% RSLogix 500 project Flip-Flop.RSS, saved by version 8.30.01.01 %
PROJECT "UNTITLED"    % processor: Bul.1763 MicroLogix 1100 Series A %

PROGRAM FILES
  LAD 2   4 rungs

DATA FILES
  O0 OUTPUT  4 elements
  I1 INPUT  6 elements
  S2 STATUS  66 elements
  B3 BINARY  1 elements
  T4 TIMER  2 elements
  C5 COUNTER  1 elements
  R6 CONTROL  1 elements
  N7 INTEGER  1 elements
  F8 FLOAT  1 elements

LADDER 2
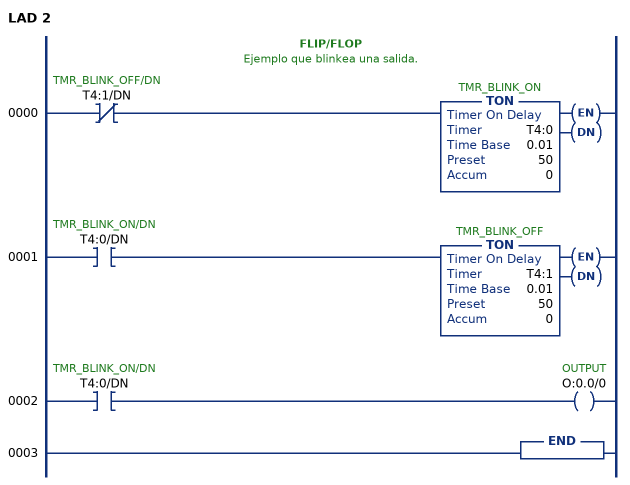
% Rung: 0 %  % edit flag set %
% TITLE: FLIP/FLOP %
% Ejemplo que blinkea una salida. %
SOR XIO T4:1/DN TON T4:0 0.01 50 0 EOR
%   T4:1  TMR_BLINK_OFF %
%   T4:0  TMR_BLINK_ON %
% Rung: 1 %  % edit flag set %
SOR XIC T4:0/DN TON T4:1 0.01 50 0 EOR
%   T4:0  TMR_BLINK_ON %
%   T4:1  TMR_BLINK_OFF %
% Rung: 2 %  % edit flag set %
SOR XIC T4:0/DN OTE O:0.0/0 EOR
%   T4:0  TMR_BLINK_ON %
%   O:0.0/0  "OUTPUT" %
% Rung: 3 %
SOR END EOR
